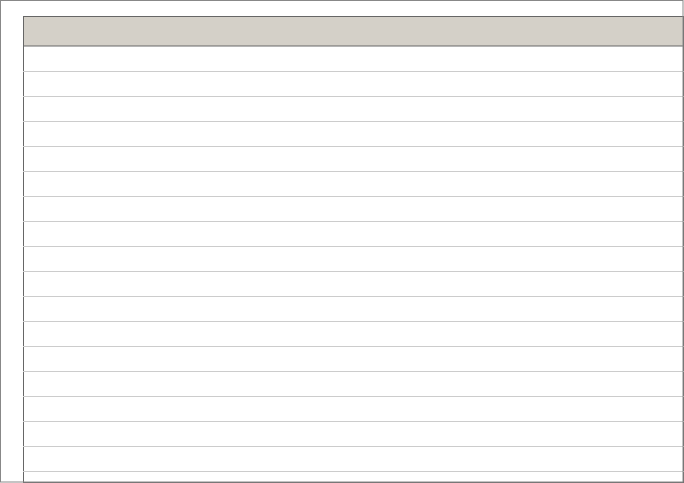
VISUALIZATION P04_Table  // 684x483
    Table (23,16 661x467), data array: Main.aryLrSin1
        p3854506369: Main.aryLrSin1[0,INDEX]
        p1892666644: Main.aryLrSin1[1,INDEX]
        p338671338: Main.aryLrSin1[2,INDEX]
        p2170511999: Main.aryLrSin1[3,INDEX]
        p3723444502: Main.aryLrSin1[4,INDEX]
        p2232123230: aryLrSin1[0]
        p511219082: aryLrSiin1[1]
        p1755163831: aryLrSin1[2]
        p4092479075: aryLrSin1[3]
        p2237128397: aryLrSin1[4]
END_VISUALIZATION

(* stored: Version 1.1.0.1, ProductVersion 3.1.4024.4
   Visu P04_Table: Id {c5593277-64ef-457c-8794-bddeb3afa9aa} *)
